// TIA Portal project "Grain Market" (V18)

(* hardware
DEVICE "S7-1200 station_1"  S7-1200 Station
   slot 0: "Rack_0"  S7-1200 Rack  Rack  V1.0
   slot 1: "PLC_1"  CPU 1214C AC/DC/Rly  6ES7 214-1BG40-0XB0  V4.6
*)

// ===== PLC "PLC_1"  CPU 1214C AC/DC/Rly =====

VAR_GLOBAL   // PLC tag table "Default tag table"
   "Start" AT %I0.0 : Bool;
   "Emergency Stop" AT %I0.1 : Bool;
   "Process" AT %M0.0 : Bool;
   "Filling Valve" AT %Q0.0 : Bool;
   "Conveyor Belt" AT %Q0.1 : Bool;
   "Start Sensor" AT %I0.2 : Bool;
   "Filled Sack Sensor" AT %I0.3 : Bool;
   "Sewing Sensor" AT %I0.4 : Bool;
   "Sewing machine" AT %Q0.2 : Bool;
END_VAR

// folder: System blocks/Program resources

DATA_BLOCK "IEC_Timer_0_DB"   // DB1
{ S7_Optimized_Access := 'TRUE' }
AUTHOR : Simatic
FAMILY : IEC
NAME : IEC_TMR
VERSION : 1.0
// stored: InstanceOfName IEC_TIMER
"IEC_TIMER"
BEGIN
END_DATA_BLOCK

// folder: (top level)

ORGANIZATION_BLOCK "Main"   // OB1, LAD, ProgramCycle
TITLE = "Main Program Sweep (Cycle)"
{ S7_Optimized_Access := 'TRUE' }
VERSION : 0.1
   VAR_INPUT
      Initial_Call : Bool;   // Initial call of this OB
      Remanence : Bool;   // =True, if remanent data are available
   END_VAR
   VAR_TEMP   // added for the SCL form of the ladder/FBD networks
      _w1 : Bool;
   END_VAR
BEGIN

REGION Network 1
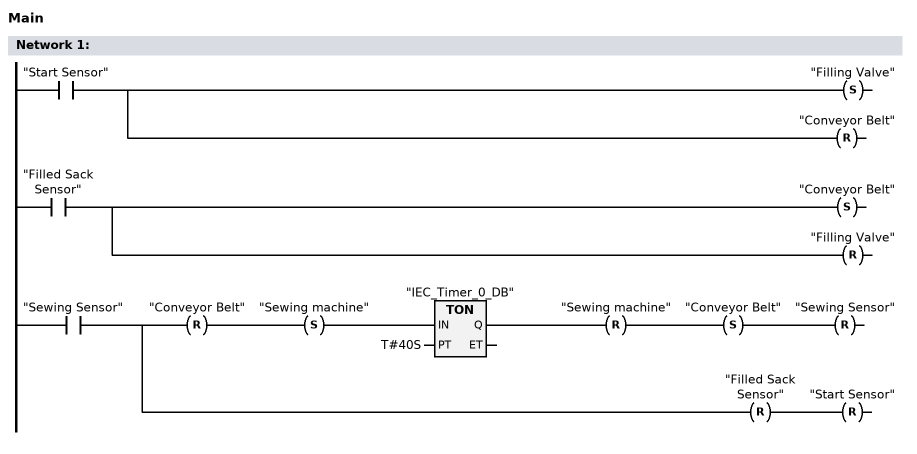
   IF "Start Sensor" THEN
       "Filling Valve" := TRUE;
       "Conveyor Belt" := FALSE;
   END_IF;
   IF "Filled Sack Sensor" THEN
       "Conveyor Belt" := TRUE;
       "Filling Valve" := FALSE;
   END_IF;
   IF "Sewing Sensor" THEN
       "Conveyor Belt" := FALSE;
       "Sewing machine" := TRUE;
   END_IF;
   "IEC_Timer_0_DB".TON(IN := "Sewing Sensor", PT := T#40S);
   IF "IEC_Timer_0_DB".Q THEN
       "Sewing machine" := FALSE;
       "Conveyor Belt" := TRUE;
   END_IF;
   #_w1 := "Sewing Sensor";
   IF "IEC_Timer_0_DB".Q THEN "Sewing Sensor" := FALSE; END_IF;
   IF #_w1 THEN
       "Filled Sack Sensor" := FALSE;
       "Start Sensor" := FALSE;
   END_IF;
END_REGION
END_ORGANIZATION_BLOCK